TYPE Vec2b : ARRAY[1..2] OF BOOL; END_TYPE

(* stored: Version 1.1.0.1, ProductVersion 3.1.4024.11
   DUT Vec2b: Id {d67e2f94-9064-4c6a-8ba8-96556083e06e} *)
